ABB RAPID module: Module1-simulacion.mod

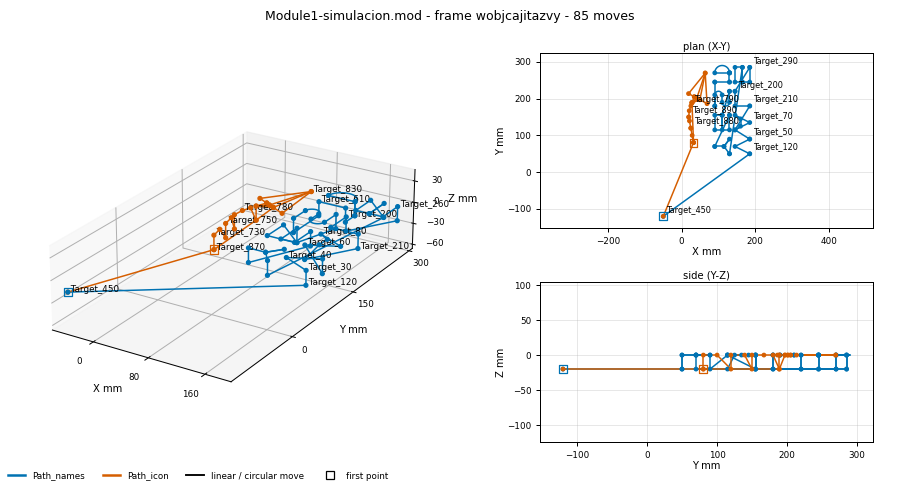
[picture p0: tool path of Module1-simulacion.mod in frame wobjcajitazvy, 85 of 87 moves have a stored position in this frame; points joined in program order, loops and branches not executed]
MODULE Module1
    CONST robtarget Target_Home:=[[602.716403522,0,579.286570049],[0.258819045,0,0.965925826,0],[0,0,0,0],[9E+09,9E+09,9E+09,9E+09,9E+09,9E+09]];
    CONST robtarget Target_10:=[[0,797.668689608,493.604548276],[0.241844763,-0.664463024,0.664463024,0.241844763],[1,0,0,0],[9E+09,9E+09,9E+09,9E+09,9E+09,9E+09]];
    CONST robtarget Target_20:=[[0,0,0],[1,0,0,0],[0,0,0,0],[9E+09,9E+09,9E+09,9E+09,9E+09,9E+09]];
    CONST robtarget Target_30:=[[185,50,0],[0,0.258819045,0,0.965925826],[-1,-1,0,0],[9E+09,9E+09,9E+09,9E+09,9E+09,9E+09]];
    CONST robtarget Target_40:=[[145,70,0],[0,0.258819045,0,0.965925826],[-1,-1,0,0],[9E+09,9E+09,9E+09,9E+09,9E+09,9E+09]];
    CONST robtarget Target_50:=[[185,90,0],[0,0.258819045,0,0.965925826],[-1,-1,0,0],[9E+09,9E+09,9E+09,9E+09,9E+09,9E+09]];
    CONST robtarget Target_130:=[[185,90,-20],[0,0.258819045,0,0.965925826],[-1,-1,0,0],[9E+09,9E+09,9E+09,9E+09,9E+09,9E+09]];
    CONST robtarget Target_120:=[[185,50,-20],[0,0.258819045,0,0.965925826],[-1,-1,0,0],[9E+09,9E+09,9E+09,9E+09,9E+09,9E+09]];
    CONST robtarget Target_450:=[[-50,-120,-20],[0,0.258819045,0,0.965925826],[0,0,0,0],[9E+09,9E+09,9E+09,9E+09,9E+09,9E+09]];
    CONST robtarget Target_60:=[[145,115,0],[0,0.258819045,0,0.965925826],[-1,-1,0,0],[9E+09,9E+09,9E+09,9E+09,9E+09,9E+09]];
    CONST robtarget Target_70:=[[185,135,0],[0,0.258819045,0,0.965925826],[-1,-1,0,0],[9E+09,9E+09,9E+09,9E+09,9E+09,9E+09]];
    CONST robtarget Target_80:=[[145,155,0],[0,0.258819045,0,0.965925826],[-1,-1,0,0],[9E+09,9E+09,9E+09,9E+09,9E+09,9E+09]];
    CONST robtarget Target_90:=[[160,145,0],[0,0.258819045,0,0.965925826],[-1,-1,0,0],[9E+09,9E+09,9E+09,9E+09,9E+09,9E+09]];
    CONST robtarget Target_100:=[[160,125,0],[0,0.258819045,0,0.965925826],[-1,-1,0,0],[9E+09,9E+09,9E+09,9E+09,9E+09,9E+09]];
    CONST robtarget Target_140:=[[145,115,-20],[0,0.258819045,0,0.965925826],[-1,-1,0,0],[9E+09,9E+09,9E+09,9E+09,9E+09,9E+09]];
    CONST robtarget Target_210:=[[185,180,-20],[0,0.258819045,0,0.965925826],[-1,-1,0,0],[9E+09,9E+09,9E+09,9E+09,9E+09,9E+09]];
    CONST robtarget Target_190:=[[185,180,0],[0,0.258819045,0,0.965925826],[-1,-1,0,0],[9E+09,9E+09,9E+09,9E+09,9E+09,9E+09]];
    CONST robtarget Target_180:=[[145,180,0],[0,0.258819045,0,0.965925826],[-1,-1,0,0],[9E+09,9E+09,9E+09,9E+09,9E+09,9E+09]];
    CONST robtarget Target_200:=[[145,220,0],[0,0.258819045,0,0.965925826],[-1,-1,0,0],[9E+09,9E+09,9E+09,9E+09,9E+09,9E+09]];
    CONST robtarget Target_220:=[[145,220,-20],[0,0.258819045,0,0.965925826],[-1,-1,0,0],[9E+09,9E+09,9E+09,9E+09,9E+09,9E+09]];
    CONST robtarget Target_290:=[[185,285,-20],[0,0.258819045,0,0.965925826],[-1,0,-1,0],[9E+09,9E+09,9E+09,9E+09,9E+09,9E+09]];
    CONST robtarget Target_260:=[[185,285,0],[0,0.258819045,0,0.965925826],[-1,0,-1,0],[9E+09,9E+09,9E+09,9E+09,9E+09,9E+09]];
    CONST robtarget Target_250:=[[185,245,0],[0,0.258819045,0,0.965925826],[-1,-1,0,0],[9E+09,9E+09,9E+09,9E+09,9E+09,9E+09]];
    CONST robtarget Target_270:=[[165,245,0],[0,0.258819045,0,0.965925826],[-1,-1,0,0],[9E+09,9E+09,9E+09,9E+09,9E+09,9E+09]];
    CONST robtarget Target_280:=[[165,285,0],[0,0.258819045,0,0.965925826],[-1,0,-1,0],[9E+09,9E+09,9E+09,9E+09,9E+09,9E+09]];
    CONST robtarget Target_230:=[[145,245,0],[0,0.258819045,0,0.965925826],[-1,-1,0,0],[9E+09,9E+09,9E+09,9E+09,9E+09,9E+09]];
    CONST robtarget Target_240:=[[145,285,0],[0,0.258819045,0,0.965925826],[-1,0,-1,0],[9E+09,9E+09,9E+09,9E+09,9E+09,9E+09]];
    CONST robtarget Target_300:=[[165,285,-20],[0,0.258819045,0,0.965925826],[-1,0,-1,0],[9E+09,9E+09,9E+09,9E+09,9E+09,9E+09]];
    CONST robtarget Target_350:=[[130,50,-20],[0,0.258819045,0,0.965925826],[-1,-1,0,0],[9E+09,9E+09,9E+09,9E+09,9E+09,9E+09]];
    CONST robtarget Target_310:=[[130,50,0],[0,0.258819045,0,0.965925826],[-1,-1,0,0],[9E+09,9E+09,9E+09,9E+09,9E+09,9E+09]];
    CONST robtarget Target_330:=[[115,70,0],[0,0.258819045,0,0.965925826],[-1,-1,0,0],[9E+09,9E+09,9E+09,9E+09,9E+09,9E+09]];
    CONST robtarget Target_320:=[[130,90,0],[0,0.258819045,0,0.965925826],[-1,-1,0,0],[9E+09,9E+09,9E+09,9E+09,9E+09,9E+09]];
    CONST robtarget Target_340:=[[90,70,0],[0,0.258819045,0,0.965925826],[-1,-1,0,0],[9E+09,9E+09,9E+09,9E+09,9E+09,9E+09]];
    CONST robtarget Target_360:=[[90,70,-20],[0,0.258819045,0,0.965925826],[-1,-1,0,0],[9E+09,9E+09,9E+09,9E+09,9E+09,9E+09]];
    CONST robtarget Target_430:=[[130,155,-20],[0,0.258819045,0,0.965925826],[-1,-1,0,0],[9E+09,9E+09,9E+09,9E+09,9E+09,9E+09]];
    CONST robtarget Target_380:=[[130,155,0],[0,0.258819045,0,0.965925826],[-1,-1,0,0],[9E+09,9E+09,9E+09,9E+09,9E+09,9E+09]];
    CONST robtarget Target_370:=[[130,115,0],[0,0.258819045,0,0.965925826],[-1,-1,0,0],[9E+09,9E+09,9E+09,9E+09,9E+09,9E+09]];
    CONST robtarget Target_410:=[[90,115,0],[0,0.258819045,0,0.965925826],[-1,-1,0,0],[9E+09,9E+09,9E+09,9E+09,9E+09,9E+09]];
    CONST robtarget Target_400:=[[90,155,0],[0,0.258819045,0,0.965925826],[-1,-1,0,0],[9E+09,9E+09,9E+09,9E+09,9E+09,9E+09]];
    CONST robtarget Target_440:=[[110,155,-20],[0,0.258819045,0,0.965925826],[-1,-1,0,0],[9E+09,9E+09,9E+09,9E+09,9E+09,9E+09]];
    CONST robtarget Target_390:=[[110,155,0],[0,0.258819045,0,0.965925826],[-1,-1,0,0],[9E+09,9E+09,9E+09,9E+09,9E+09,9E+09]];
    CONST robtarget Target_420:=[[110,115,0],[0,0.258819045,0,0.965925826],[-1,-1,0,0],[9E+09,9E+09,9E+09,9E+09,9E+09,9E+09]];
    CONST robtarget Target_480:=[[130,180,0],[1,0,0,0],[0,0,0,0],[9E+09,9E+09,9E+09,9E+09,9E+09,9E+09]];
    CONST robtarget Target_500:=[[130,220,0],[0,0.258819045,0,0.965925826],[-1,-1,0,0],[9E+09,9E+09,9E+09,9E+09,9E+09,9E+09]];
    CONST robtarget Target_530:=[[110,190,0],[0,0.258819045,0,0.965925826],[-1,-1,0,0],[9E+09,9E+09,9E+09,9E+09,9E+09,9E+09]];
    CONST robtarget Target_540:=[[130,190,0],[0,0.258819045,0,0.965925826],[-1,-1,0,0],[9E+09,9E+09,9E+09,9E+09,9E+09,9E+09]];
    CONST robtarget Target_520:=[[120,180,0],[0,0.258819045,0,0.965925826],[-1,-1,0,0],[9E+09,9E+09,9E+09,9E+09,9E+09,9E+09]];
    CONST robtarget Target_580:=[[130,220,-20],[0,0.258819045,0,0.965925826],[-1,-1,0,0],[9E+09,9E+09,9E+09,9E+09,9E+09,9E+09]];
    CONST robtarget Target_550:=[[110,210,0],[0,0.258819045,0,0.965925826],[-1,-1,0,0],[9E+09,9E+09,9E+09,9E+09,9E+09,9E+09]];
    CONST robtarget Target_560:=[[100,220,0],[0,0.258819045,0,0.965925826],[-1,-1,0,0],[9E+09,9E+09,9E+09,9E+09,9E+09,9E+09]];
    CONST robtarget Target_570:=[[90,210,0],[0,0.258819045,0,0.965925826],[-1,-1,0,0],[9E+09,9E+09,9E+09,9E+09,9E+09,9E+09]];
    CONST robtarget Target_490:=[[90,180,0],[0,0.258819045,0,0.965925826],[-1,-1,0,0],[9E+09,9E+09,9E+09,9E+09,9E+09,9E+09]];
    CONST robtarget Target_590:=[[90,180,-20],[0,0.258819045,0,0.965925826],[-1,-1,0,0],[9E+09,9E+09,9E+09,9E+09,9E+09,9E+09]];
    CONST robtarget Target_660:=[[90,245,-20],[0,0.258819045,0,0.965925826],[-1,-1,0,0],[9E+09,9E+09,9E+09,9E+09,9E+09,9E+09]];
    CONST robtarget Target_610:=[[90,245,0],[0,0.258819045,0,0.965925826],[-1,-1,0,0],[9E+09,9E+09,9E+09,9E+09,9E+09,9E+09]];
    CONST robtarget Target_600:=[[130,245,0],[0,0.258819045,0,0.965925826],[-1,-1,0,0],[9E+09,9E+09,9E+09,9E+09,9E+09,9E+09]];
    CONST robtarget Target_650:=[[130,245,-20],[0,0.258819045,0,0.965925826],[-1,-1,0,0],[9E+09,9E+09,9E+09,9E+09,9E+09,9E+09]];
    CONST robtarget Target_680:=[[130,270,-20],[0,0.258819045,0,0.965925826],[-1,0,0,0],[9E+09,9E+09,9E+09,9E+09,9E+09,9E+09]];
    CONST robtarget Target_620:=[[130,270,0],[0,0.258819045,0,0.965925826],[-1,0,0,0],[9E+09,9E+09,9E+09,9E+09,9E+09,9E+09]];
    CONST robtarget Target_640:=[[110,290,0],[0,0.258819045,0,0.965925826],[-2,0,-1,0],[9E+09,9E+09,9E+09,9E+09,9E+09,9E+09]];
    CONST robtarget Target_630:=[[90,270,0],[0,0.258819045,0,0.965925826],[-1,0,0,0],[9E+09,9E+09,9E+09,9E+09,9E+09,9E+09]];
    CONST robtarget Target_870:=[[32.223,80.467,-20],[0,0,0,1],[0,0,0,0],[9E+09,9E+09,9E+09,9E+09,9E+09,9E+09]];
    CONST robtarget Target_730:=[[32.223,80.467,0],[0,0,0,1],[-1,-1,0,0],[9E+09,9E+09,9E+09,9E+09,9E+09,9E+09]];
    CONST robtarget Target_740:=[[28.538,100.125,0],[0,0,0,1],[-1,-1,0,0],[9E+09,9E+09,9E+09,9E+09,9E+09,9E+09]];
    CONST robtarget Target_880:=[[24.853,119.783,-20],[0,0,0,1],[-1,-1,0,0],[9E+09,9E+09,9E+09,9E+09,9E+09,9E+09]];
    CONST robtarget Target_750:=[[24.853,119.783,0],[0,0,0,1],[-1,-1,0,0],[9E+09,9E+09,9E+09,9E+09,9E+09,9E+09]];
    CONST robtarget Target_760:=[[21.169,139.44,0],[0,0,0,1],[-1,-1,0,0],[9E+09,9E+09,9E+09,9E+09,9E+09,9E+09]];
    CONST robtarget Target_890:=[[19.22,149.833,-20],[0,0,0,1],[-1,-1,0,0],[9E+09,9E+09,9E+09,9E+09,9E+09,9E+09]];
    CONST robtarget Target_770:=[[19.22,149.833,0],[0,0,0,1],[-1,-1,0,0],[9E+09,9E+09,9E+09,9E+09,9E+09,9E+09]];
    CONST robtarget Target_780:=[[20.586,167,0],[0,0,0,1],[-1,-1,0,0],[9E+09,9E+09,9E+09,9E+09,9E+09,9E+09]];
    CONST robtarget Target_790:=[[25,180,0],[0,0,0,1],[-1,-1,0,0],[9E+09,9E+09,9E+09,9E+09,9E+09,9E+09]];
    CONST robtarget Target_900:=[[28,189,-20],[0,0,0,1],[-1,-1,0,0],[9E+09,9E+09,9E+09,9E+09,9E+09,9E+09]];
    CONST robtarget Target_800:=[[28,189,0],[0,0,0,1],[-1,-1,0,0],[9E+09,9E+09,9E+09,9E+09,9E+09,9E+09]];
    CONST robtarget Target_810:=[[49.5,197,0],[0,0,0,1],[-1,-1,0,0],[9E+09,9E+09,9E+09,9E+09,9E+09,9E+09]];
    CONST robtarget Target_820:=[[68.98,186.28,0],[0,0,0,1],[-1,-1,0,0],[9E+09,9E+09,9E+09,9E+09,9E+09,9E+09]];
    CONST robtarget Target_830:=[[64,269.5,0],[0,0,0,1],[-1,0,0,0],[9E+09,9E+09,9E+09,9E+09,9E+09,9E+09]];
    CONST robtarget Target_840:=[[18.71,213.6,0],[0,0,0,1],[-1,-1,0,0],[9E+09,9E+09,9E+09,9E+09,9E+09,9E+09]];
    CONST robtarget Target_850:=[[34.34,205.06,0],[0,0,0,1],[-1,-1,0,0],[9E+09,9E+09,9E+09,9E+09,9E+09,9E+09]];
    CONST robtarget Target_860:=[[41,201,0],[0,0,0,1],[-1,-1,0,0],[9E+09,9E+09,9E+09,9E+09,9E+09,9E+09]];
    PROC Path_home()
        MoveJ Target_Home,v100,z10,MyNewTool\WObj:=wobj0;
    ENDPROC

    PROC main()
        SetDO DO_01, 0;
        SetDO DO_02, 0;
        SetDO DO_03, 0;
        WHILE TRUE DO
        Path_home;
            IF DI_01=1 THEN
                Set DO_01;  !la banda transporta el pastel a la posición donde se hace el decorado
                WaitTime 4; !tiempo de espera mientras la banda transporta el pastel a la posición posición donde se hace el decorado
                Path_names; !se hacen los trazos para hacer los nombres de los miembros del equipo
                Path_icon;  !se hacen los trazos para hacer un ícono
                WaitTime 2; !tiempo de espera por seguridad
                Path_home;  !el robot vuelve a home
                Reset DO_01;
                Set DO_01; !la banda transporta el pastel fuera de la posición donde se hace el decorado
                Reset DO_01;
                WaitUntil DI_01=0;
            ENDIF


            IF DI_02=1 THEN
                Set DO_02;
                Path_maintenance;!el robot va a la posición de mantenimiento donde se hace el montaje de la herramienta
                Reset DO_02;
                WaitUntil DI_02=0; !se espera hasta que el estudiante coloque o desmonte la herramienta y posteriormente, uno mismo cambia el valor de la entrada
                Path_home; !retorna a home
            ENDIF

            IF DI_03=1 THEN
                Set DO_03; !La banda transporta el pastel a un extremo de la banda
                Reset DO_03;
                WaitUntil DI_03=0;
            ENDIF

        ENDWHILE
    ENDPROC

    PROC Path_maintenance()
        MoveJ Target_10,v100,z10,MyNewTool\WObj:=wobj0;
    ENDPROC
    PROC Path_names()
        MoveJ Target_450,v100,z10,MyNewTool\WObj:=wobjcajitazvy;
        MoveL Target_120,v100,z10,MyNewTool\WObj:=wobjcajitazvy;
        MoveL Target_30,v100,z10,MyNewTool\WObj:=wobjcajitazvy;
        MoveL Target_40,v100,z10,MyNewTool\WObj:=wobjcajitazvy;
        MoveL Target_50,v100,z10,MyNewTool\WObj:=wobjcajitazvy;
        MoveL Target_130,v100,z10,MyNewTool\WObj:=wobjcajitazvy;
        MoveL Target_60,v100,z10,MyNewTool\WObj:=wobjcajitazvy;
        MoveL Target_70,v100,z10,MyNewTool\WObj:=wobjcajitazvy;
        MoveL Target_80,v100,z10,MyNewTool\WObj:=wobjcajitazvy;
        MoveL Target_90,v100,z10,MyNewTool\WObj:=wobjcajitazvy;
        MoveL Target_100,v100,z10,MyNewTool\WObj:=wobjcajitazvy;
        MoveL Target_140,v100,z10,MyNewTool\WObj:=wobjcajitazvy;
        MoveL Target_210,v100,z10,MyNewTool\WObj:=wobjcajitazvy;
        MoveL Target_190,v100,z10,MyNewTool\WObj:=wobjcajitazvy;
        MoveL Target_180,v100,z10,MyNewTool\WObj:=wobjcajitazvy;
        MoveL Target_200,v100,z10,MyNewTool\WObj:=wobjcajitazvy;
        MoveL Target_220,v100,z10,MyNewTool\WObj:=wobjcajitazvy;
        MoveL Target_290,v100,z10,MyNewTool\WObj:=wobjcajitazvy;
        MoveL Target_260,v100,z10,MyNewTool\WObj:=wobjcajitazvy;
        MoveL Target_250,v100,z10,MyNewTool\WObj:=wobjcajitazvy;
        MoveL Target_270,v100,z10,MyNewTool\WObj:=wobjcajitazvy;
        MoveL Target_280,v100,z10,MyNewTool\WObj:=wobjcajitazvy;
        MoveL Target_270,v100,z10,MyNewTool\WObj:=wobjcajitazvy;
        MoveL Target_230,v100,z10,MyNewTool\WObj:=wobjcajitazvy;
        MoveL Target_240,v100,z10,MyNewTool\WObj:=wobjcajitazvy;
        MoveL Target_300,v100,z10,MyNewTool\WObj:=wobjcajitazvy;
        MoveL Target_350,v100,z10,MyNewTool\WObj:=wobjcajitazvy;
        MoveL Target_310,v100,z10,MyNewTool\WObj:=wobjcajitazvy;
        MoveL Target_330,v100,z10,MyNewTool\WObj:=wobjcajitazvy;
        MoveL Target_320,v100,z10,MyNewTool\WObj:=wobjcajitazvy;
        MoveL Target_330,v100,z10,MyNewTool\WObj:=wobjcajitazvy;
        MoveL Target_340,v100,z10,MyNewTool\WObj:=wobjcajitazvy;
        MoveL Target_360,v100,z10,MyNewTool\WObj:=wobjcajitazvy;
        MoveL Target_430,v100,z10,MyNewTool\WObj:=wobjcajitazvy;
        MoveL Target_380,v100,z10,MyNewTool\WObj:=wobjcajitazvy;
        MoveL Target_370,v100,z10,MyNewTool\WObj:=wobjcajitazvy;
        MoveL Target_410,v100,z10,MyNewTool\WObj:=wobjcajitazvy;
        MoveL Target_400,v100,z10,MyNewTool\WObj:=wobjcajitazvy;
        MoveL Target_440,v100,z10,MyNewTool\WObj:=wobjcajitazvy;
        MoveL Target_390,v100,z10,MyNewTool\WObj:=wobjcajitazvy;
        MoveL Target_420,v100,z10,MyNewTool\WObj:=wobjcajitazvy;
        MoveL Target_440,v100,z10,MyNewTool\WObj:=wobjcajitazvy;
        MoveL Target_580,v100,z10,MyNewTool\WObj:=wobjcajitazvy;
        MoveL Target_500,v100,z10,MyNewTool\WObj:=wobjcajitazvy;
        MoveL Target_540,v100,z10,MyNewTool\WObj:=wobjcajitazvy;
        MoveC Target_520,Target_530,v100,z10,MyNewTool\WObj:=wobjcajitazvy;
        MoveL Target_550,v100,z10,MyNewTool\WObj:=wobjcajitazvy;
        MoveC Target_560,Target_570,v100,z10,MyNewTool\WObj:=wobjcajitazvy;
        MoveL Target_490,v100,z10,MyNewTool\WObj:=wobjcajitazvy;
        MoveL Target_590,v100,z10,MyNewTool\WObj:=wobjcajitazvy;
        MoveL Target_660,v100,z10,MyNewTool\WObj:=wobjcajitazvy;
        MoveL Target_610,v100,z10,MyNewTool\WObj:=wobjcajitazvy;
        MoveL Target_600,v100,z10,MyNewTool\WObj:=wobjcajitazvy;
        MoveL Target_650,v100,z10,MyNewTool\WObj:=wobjcajitazvy;
        MoveL Target_680,v100,z10,MyNewTool\WObj:=wobjcajitazvy;
        MoveL Target_620,v100,z10,MyNewTool\WObj:=wobjcajitazvy;
        MoveC Target_640,Target_630,v100,z10,MyNewTool\WObj:=wobjcajitazvy;
        MoveL Target_620,v100,z10,MyNewTool\WObj:=wobjcajitazvy;
        MoveL Target_680,v100,z10,MyNewTool\WObj:=wobjcajitazvy;
    ENDPROC
    PROC Path_icon()
        MoveL Target_870,v100,z10,MyNewTool\WObj:=wobjcajitazvy;
        MoveL Target_730,v100,z10,MyNewTool\WObj:=wobjcajitazvy;
        MoveL Target_740,v100,z10,MyNewTool\WObj:=wobjcajitazvy;
        MoveL Target_880,v100,z10,MyNewTool\WObj:=wobjcajitazvy;
        MoveL Target_750,v100,z10,MyNewTool\WObj:=wobjcajitazvy;
        MoveL Target_760,v100,z10,MyNewTool\WObj:=wobjcajitazvy;
        MoveL Target_890,v100,z10,MyNewTool\WObj:=wobjcajitazvy;
        MoveL Target_770,v100,z10,MyNewTool\WObj:=wobjcajitazvy;
        MoveL Target_780,v100,z10,MyNewTool\WObj:=wobjcajitazvy;
        MoveL Target_790,v100,z10,MyNewTool\WObj:=wobjcajitazvy;
        MoveL Target_900,v100,z10,MyNewTool\WObj:=wobjcajitazvy;
        MoveL Target_800,v100,z10,MyNewTool\WObj:=wobjcajitazvy;
        MoveL Target_810,v100,z10,MyNewTool\WObj:=wobjcajitazvy;
        MoveL Target_820,v100,z10,MyNewTool\WObj:=wobjcajitazvy;
        MoveL Target_830,v100,z10,MyNewTool\WObj:=wobjcajitazvy;
        MoveL Target_840,v100,z10,MyNewTool\WObj:=wobjcajitazvy;
        MoveL Target_850,v100,z10,MyNewTool\WObj:=wobjcajitazvy;
        MoveL Target_860,v100,z10,MyNewTool\WObj:=wobjcajitazvy;
        MoveL Target_800,v100,z10,MyNewTool\WObj:=wobjcajitazvy;
        MoveL Target_850,v100,z10,MyNewTool\WObj:=wobjcajitazvy;
        MoveL Target_860,v100,z10,MyNewTool\WObj:=wobjcajitazvy;
        MoveL Target_830,v100,z10,MyNewTool\WObj:=wobjcajitazvy;
        MoveL Target_810,v100,z10,MyNewTool\WObj:=wobjcajitazvy;
        MoveL Target_900,v100,z10,MyNewTool\WObj:=wobjcajitazvy;
        MoveL Target_870,v100,z10,MyNewTool\WObj:=wobjcajitazvy;
        MoveL Target_450,v100,z10,MyNewTool\WObj:=wobjcajitazvy;
    ENDPROC
ENDMODULE
